# EPICS autosave request: iocBoot/sioc-esb-xps3/xps.req
file xpsm.req P=ESB:XPS3:m1
file xpsm.req P=ESB:XPS3:m2
file xpsm.req P=ESB:XPS3:m3
file xpsm.req P=ESB:XPS3:m4
file xpsm.req P=ESB:XPS3:m5
file xpsm.req P=ESB:XPS3:m6
file xpsm.req P=ESB:XPS3:m7
file xpsm.req P=ESB:XPS3:m8
